(* IEC 61131-3 sources: finder/src/Ar/finder, 3 files *)

(* ---- Types.typ ---- *)
(*
 * File: Types.typ
 * Copyright (c) 2023 Loupe
 * https://loupe.team
 *
 * This file is part of Finder, licensed under the MIT License.
 *)

TYPE
	finder_typ : 	STRUCT
		in : finderIn_typ;
		out : finderOut_typ;
		internal : finderInternal_typ;
	END_STRUCT;
	finderIn_typ : 	STRUCT
		filedevice : STRING[80];
		cwd : STRING[240];
		refresh : BOOL;
	END_STRUCT;
	finderOut_typ : 	STRUCT
		done : BOOL;
		updating : BOOL;
		status : UDINT;
	END_STRUCT;
	finderInternal_typ : 	STRUCT
		path : STRING[240];
		cwd : STRING[240];
		state : INT;
		ident : UDINT;
		directoryOpen : DirOpen;
		directoryRead : DirReadEx;
		directoryClose : DirClose;
		dirData : fiDIR_READ_EX_DATA;
		obj : REFERENCE TO UDINT;
		comma : BOOL;
	END_STRUCT;
END_TYPE

(* ---- Finder.fun ---- *)
(*
 * File: Finder.fun
 * Copyright (c) 2023 Loupe
 * https://loupe.team
 *
 * This file is part of Finder, licensed under the MIT License.
 *)

FUNCTION finder : USINT
	VAR_INPUT
		in : finder_typ;
		pBuf : UDINT;
		sBuf : UDINT;
	END_VAR
END_FUNCTION

(* ---- Constants.var ---- *)
(*
 * File: Constants.var
 * Copyright (c) 2023 Loupe
 * https://loupe.team
 *
 * This file is part of Finder, licensed under the MIT License.
 *)

VAR CONSTANT

END_VAR
